// Mitsubishi GX Works2 project: 6   PLC: FX3U/FX3UC

PROGRAM MAIN
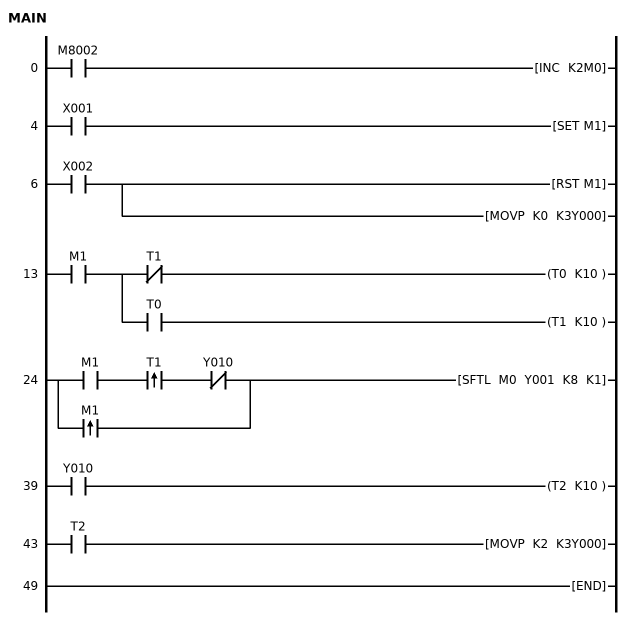
0     LD      M8002
      INC     K2M0
4     LD      X001
      SET     M1
6     LD      X002
      RST     M1
      MOVP    K0 K3Y000
13    LD      M1
      MPS
      ANI     T1
      OUT     T0 K10
      MPP
      AND     T0
      OUT     T1 K10
24    LD      M1
      ANDP    T1
      ANI     Y010
      ORP     M1
      SFTL    M0 Y001 K8 K1
39    LD      Y010
      OUT     T2 K10
43    LD      T2
      MOVP    K2 K3Y000
49    END
END_PROGRAM
